FUNCTION_BLOCK PAEActValve3 EXTENDS PAEActuator3way
VAR_INPUT
END_VAR
VAR_OUTPUT
END_VAR
VAR
END_VAR

END_FUNCTION_BLOCK

(* stored: Version 1.1.0.1, ProductVersion 3.1.4020.12
   POU PAEActValve3: Id {e6651301-b59d-4be3-8af8-554efbcae8cf}, SpecialFunc None *)
